// TIA Portal V20 export
FUNCTION_BLOCK "Sensors"   // FB505, FBD
{ S7_Optimized_Access := 'TRUE' }
// stored: AutoNumber false, MemoryReserve 100, SetENOAutomatically false
   VAR
      Var { ExternalAccessible := 'False'; ExternalVisible := 'False'; ExternalWritable := 'False'} : "TypeVar";
      Enc { ExternalAccessible := 'False'; ExternalVisible := 'False'; ExternalWritable := 'False'} : Array[1..3] of "SysCounterFast";
      S { ExternalAccessible := 'False'; ExternalVisible := 'False'; ExternalWritable := 'False'} : Array[1..5] of "SysSensor";
      SIO { ExternalAccessible := 'False'; ExternalVisible := 'False'; ExternalWritable := 'False'} : Array[1..3] of "SysWenglorP3PC301";
      senRightEncAct { ExternalAccessible := 'False'; ExternalVisible := 'False'; ExternalWritable := 'False'} : Real;
      senRightValSmoth { ExternalAccessible := 'False'; ExternalVisible := 'False'; ExternalWritable := 'False'} : Real;
      senRightCntr { ExternalAccessible := 'False'; ExternalVisible := 'False'; ExternalWritable := 'False'} : DInt;
      senRightSum { ExternalAccessible := 'False'; ExternalVisible := 'False'; ExternalWritable := 'False'} : Real;
      senLeftEncAct { ExternalAccessible := 'False'; ExternalVisible := 'False'; ExternalWritable := 'False'} : Real;
      senLeftValSmoth { ExternalAccessible := 'False'; ExternalVisible := 'False'; ExternalWritable := 'False'} : Real;
      senLeftCntr { ExternalAccessible := 'False'; ExternalVisible := 'False'; ExternalWritable := 'False'} : DInt;
      senLeftSum { ExternalAccessible := 'False'; ExternalVisible := 'False'; ExternalWritable := 'False'} : Real;
      senTopEncAct { ExternalAccessible := 'False'; ExternalVisible := 'False'; ExternalWritable := 'False'} : Real;
      senTopValSmoth { ExternalAccessible := 'False'; ExternalVisible := 'False'; ExternalWritable := 'False'} : Real;
      senTopCntr { ExternalAccessible := 'False'; ExternalVisible := 'False'; ExternalWritable := 'False'} : DInt;
      senTopSum { ExternalAccessible := 'False'; ExternalVisible := 'False'; ExternalWritable := 'False'} : Real;
      deltaSaved { ExternalAccessible := 'False'; ExternalVisible := 'False'; ExternalWritable := 'False'} : Real;
      senLeftValValid { ExternalAccessible := 'False'; ExternalVisible := 'False'; ExternalWritable := 'False'} : Bool;
      senRightValValid { ExternalAccessible := 'False'; ExternalVisible := 'False'; ExternalWritable := 'False'} : Bool;
      senTopValValid { ExternalAccessible := 'False'; ExternalVisible := 'False'; ExternalWritable := 'False'} : Bool;
      widthMeasureOk { ExternalAccessible := 'False'; ExternalVisible := 'False'; ExternalWritable := 'False'} : Bool;
   END_VAR
   VAR_TEMP
      tempMin : Real;
      tempMax : Real;
      tempWidth : Real;
   END_VAR
   VAR_TEMP   // added for the SCL form of the ladder/FBD networks
      _w1 : Bool;
   END_VAR
BEGIN

REGION Network 1: encoder infeed scanner
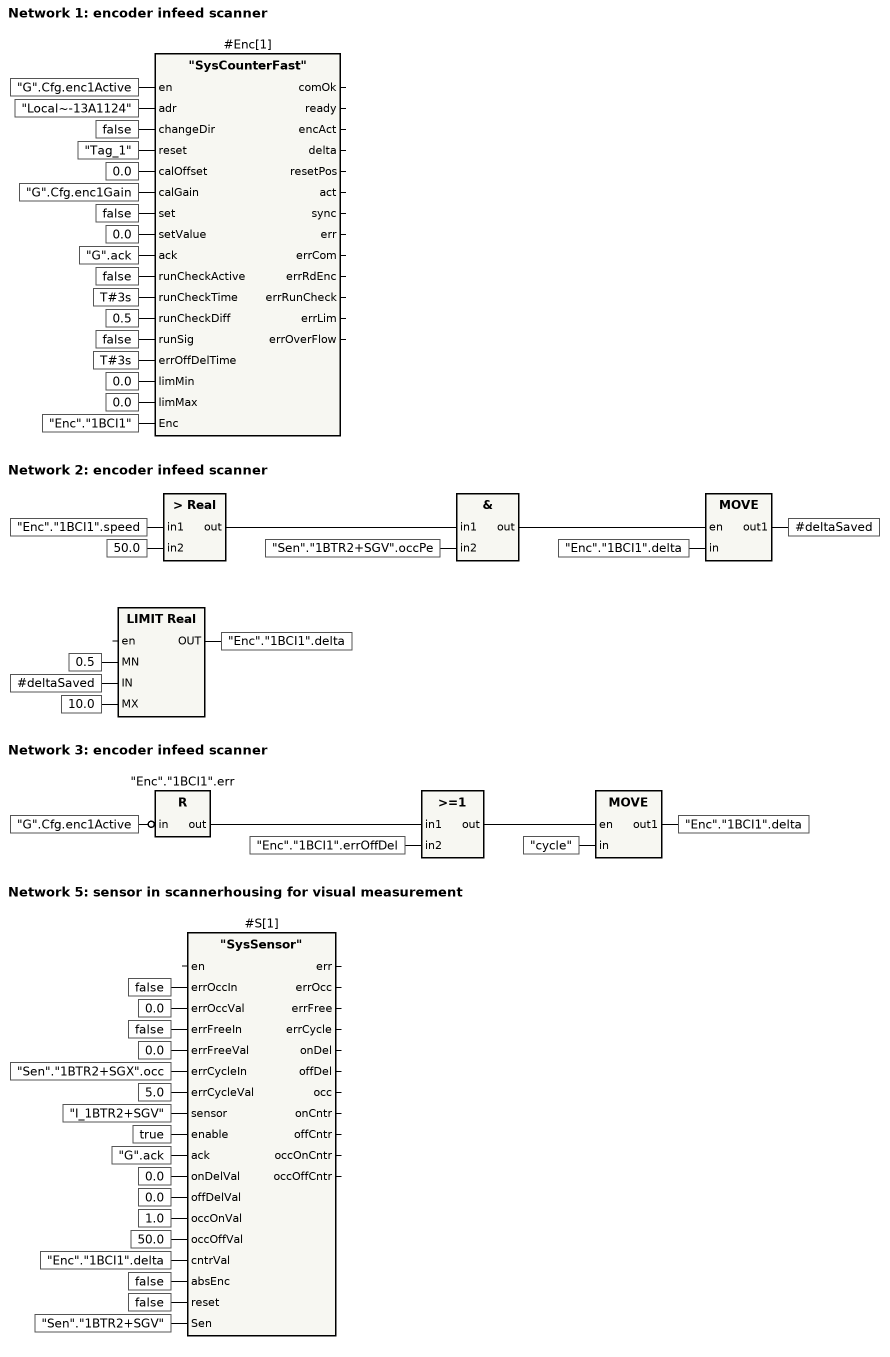
   IF "G".Cfg.enc1Active THEN
       #Enc[1](adr := "Local~-13A1124",   // "SysCounterFast"
               changeDir := false,
               reset := "Tag_1",
               calOffset := 0.0,
               calGain := "G".Cfg.enc1Gain,
               set := false,
               setValue := 0.0,
               ack := "G".ack,
               runCheckActive := false,
               runCheckTime := T#3s,
               runCheckDiff := 0.5,
               runSig := false,
               errOffDelTime := T#3s,
               limMin := 0.0,
               limMax := 0.0,
               Enc := "Enc"."1BCI1");
   END_IF;
END_REGION

REGION Network 2: encoder infeed scanner
   IF ("Enc"."1BCI1".speed > 50.0) AND "Sen"."1BTR2+SGV".occPe THEN
       #deltaSaved := "Enc"."1BCI1".delta;
   END_IF;
   "Enc"."1BCI1".delta := LIMIT(MN := 0.5, IN := #deltaSaved, MX := 10.0);
END_REGION

REGION Network 3: encoder infeed scanner
   IF NOT "G".Cfg.enc1Active THEN "Enc"."1BCI1".err := FALSE; END_IF;
   IF NOT "G".Cfg.enc1Active OR "Enc"."1BCI1".errOffDel THEN "Enc"."1BCI1".delta := "cycle"; END_IF;
END_REGION

REGION Network 4: - sensor monitoring -
END_REGION

REGION Network 5: sensor in scannerhousing for visual measurement
   #S[1](errOccIn := false,   // "SysSensor"
         errOccVal := 0.0,
         errFreeIn := false,
         errFreeVal := 0.0,
         errCycleIn := "Sen"."1BTR2+SGX".occ,
         errCycleVal := 5.0,
         sensor := "I_1BTR2+SGV",
         enable := true,
         ack := "G".ack,
         onDelVal := 0.0,
         offDelVal := 0.0,
         occOnVal := 1.0,
         occOffVal := 50.0,
         cntrVal := "Enc"."1BCI1".delta,
         absEnc := false,
         reset := false,
         Sen := "Sen"."1BTR2+SGV");
END_REGION

REGION Network 6: sensor in scannerhousing for xray measurement
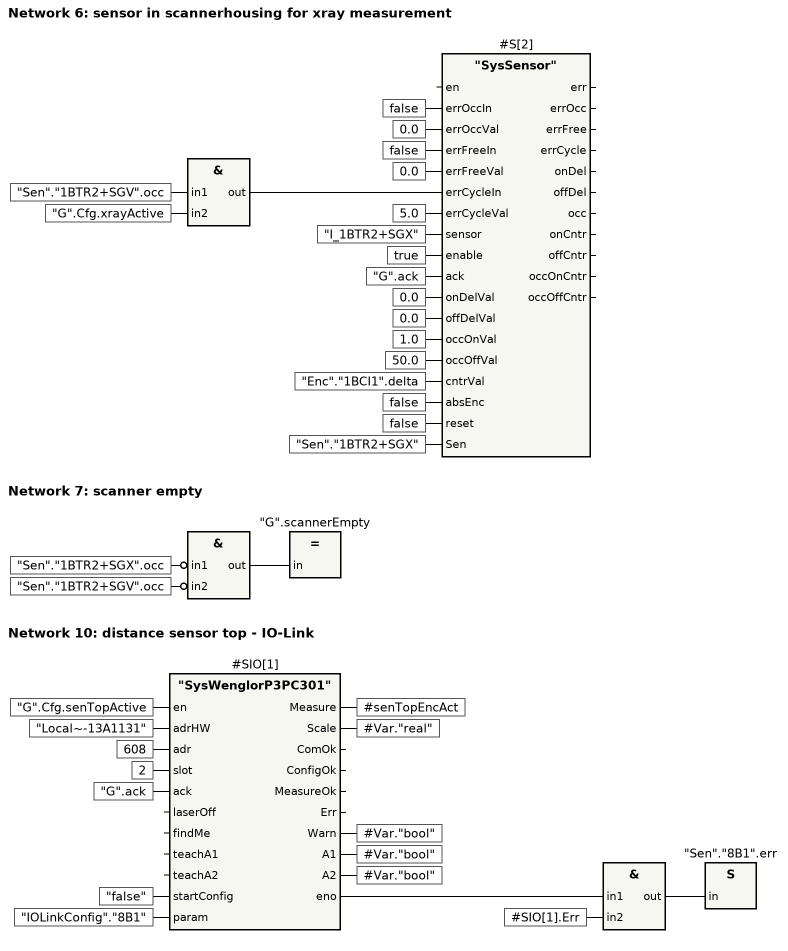
   #S[2](errOccIn := false,   // "SysSensor"
         errOccVal := 0.0,
         errFreeIn := false,
         errFreeVal := 0.0,
         errCycleIn := "Sen"."1BTR2+SGV".occ AND "G".Cfg.xrayActive,
         errCycleVal := 5.0,
         sensor := "I_1BTR2+SGX",
         enable := true,
         ack := "G".ack,
         onDelVal := 0.0,
         offDelVal := 0.0,
         occOnVal := 1.0,
         occOffVal := 50.0,
         cntrVal := "Enc"."1BCI1".delta,
         absEnc := false,
         reset := false,
         Sen := "Sen"."1BTR2+SGX");
END_REGION

REGION Network 7: scanner empty
   "G".scannerEmpty := NOT "Sen"."1BTR2+SGX".occ AND NOT "Sen"."1BTR2+SGV".occ;
END_REGION

REGION Network 8: distance sensor top
END_REGION

REGION Network 9 (SCL): distance sensor top - calibration value from pc
   "ComSd".Data.Measure.SetCalibratePosTopOk := FALSE;

   IF "ComRd".Data.Measure.SetCalibratePosTop THEN

       "Ref".senTopCalOffset := #senTopEncAct + "G".Batch.thickness;
       "ComSd".Data.Measure.SetCalibratePosTopOk := TRUE;
   END_IF;
END_REGION

REGION Network 10: distance sensor top - IO-Link
   #SIO[1](EN := "G".Cfg.senTopActive,   // "SysWenglorP3PC301"
           adrHW := "Local~-13A1131",
           adr := 608,
           slot := 2,
           ack := "G".ack,
           startConfig := "false",
           param := "IOLinkConfig"."8B1",
           Measure => #senTopEncAct,
           Scale => #Var."real",
           Warn => #Var."bool",
           A1 => #Var."bool",
           A2 => #Var."bool",
           ENO => #_w1);
   IF #_w1 AND #SIO[1].Err THEN "Sen"."8B1".err := TRUE; END_IF;
END_REGION

REGION Network 11 (SCL): distance sensor top - values
   IF "G".Cfg.senTopActive THEN
       IF #SIO[1].MeasureOk THEN
           "Sen"."8B1".val := "Ref".senTopCalOffset - #senTopEncAct;
       ELSE
           "Sen"."8B1".val := -50.0;
       END_IF;
       "ComSd".Data.Measure.ActValueTop := REAL_TO_DINT(#senTopEncAct * 10.0);

       IF "G".Cfg.modeBoardPassing = 3 THEN
           #tempMin := "G".Batch.widthMin / 4.0;
           #tempMax := "G".Batch.widthMax + 50.0;
       ELSE
           #tempMin := "G".Batch.widthMin / 2.0;
           #tempMax := "G".Batch.widthMax + 50.0;
       END_IF;
   ELSE
       #senTopEncAct :=  "Sen"."8B1".val := 0.0;
       "ComSd".Data.Measure.ActValueTop := 0;
   END_IF;
END_REGION

REGION Network 12: distance sensor top - occupied
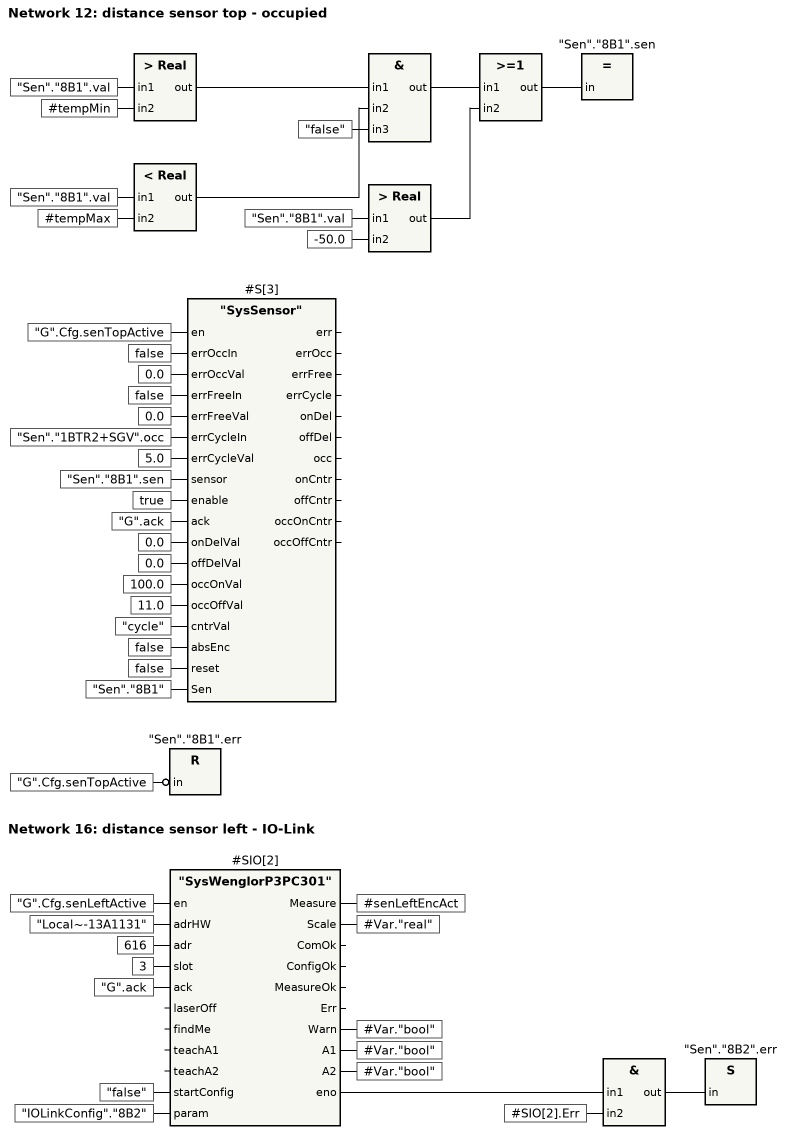
   "Sen"."8B1".sen := (("Sen"."8B1".val > #tempMin) AND ("Sen"."8B1".val < #tempMax) AND "false") OR ("Sen"."8B1".val > (-50.0));
   IF "G".Cfg.senTopActive THEN
       #S[3](errOccIn := false,   // "SysSensor"
             errOccVal := 0.0,
             errFreeIn := false,
             errFreeVal := 0.0,
             errCycleIn := "Sen"."1BTR2+SGV".occ,
             errCycleVal := 5.0,
             sensor := "Sen"."8B1".sen,
             enable := true,
             ack := "G".ack,
             onDelVal := 0.0,
             offDelVal := 0.0,
             occOnVal := 100.0,
             occOffVal := 11.0,
             cntrVal := "cycle",
             absEnc := false,
             reset := false,
             Sen := "Sen"."8B1");
   END_IF;
   IF NOT "G".Cfg.senTopActive THEN "Sen"."8B1".err := FALSE; END_IF;
END_REGION

REGION Network 13 (SCL): distance sensor top - smoothed value
   IF "Sen"."8B1".occPe THEN
       #senTopCntr := 10;
       #senTopSum := 0.0;
       #senTopValValid := false;
   ELSIF NOT "Sen"."8B1".occ OR #senTopCntr > 10 THEN
       #senTopCntr := 0;
   END_IF;

   IF "Sen"."8B1".occNe THEN
       #senTopValValid := false;
   END_IF;

   IF #senTopCntr > 0 AND "Sen"."8B1".sen THEN
       #senTopSum += "Sen"."8B1".val;
       #senTopCntr -= 1;
       IF #senTopCntr = 0 THEN
           #senTopValSmoth := #senTopSum / 10.0;
           #senTopValValid := true;
       END_IF;
   END_IF;

   IF "ComRd".Data.status.Auto AND  "G".Cfg.senTopActive THEN
       "Sen"."8B1".val := #senTopValSmoth;
   END_IF;
END_REGION

REGION Network 14: distance sensor left
END_REGION

REGION Network 15 (SCL): distance sensor left - calibration value from pc
   "ComSd".Data.Measure.SetCalibratePosLeftOk := FALSE;

   IF "ComRd".Data.Measure.SetCalibratePosLeft THEN

       #tempWidth := "G".Batch.width;
       IF "G".Cfg.modeBoardPassing = 3 THEN
           #tempWidth := "G".Batch.width / 2.0;
       END_IF;
       "Ref".senLeftCalOffset := #senLeftEncAct + #tempWidth;

       "ComSd".Data.Measure.SetCalibratePosLeftOk := TRUE;
   END_IF;
END_REGION

REGION Network 16: distance sensor left - IO-Link
   #SIO[2](EN := "G".Cfg.senLeftActive,   // "SysWenglorP3PC301"
           adrHW := "Local~-13A1131",
           adr := 616,
           slot := 3,
           ack := "G".ack,
           startConfig := "false",
           param := "IOLinkConfig"."8B2",
           Measure => #senLeftEncAct,
           Scale => #Var."real",
           Warn => #Var."bool",
           A1 => #Var."bool",
           A2 => #Var."bool",
           ENO => #_w1);
   IF #_w1 AND #SIO[2].Err THEN "Sen"."8B2".err := TRUE; END_IF;
END_REGION

REGION Network 17 (SCL): distance sensor left - values
   IF "G".Cfg.senLeftActive THEN

       IF #SIO[2].MeasureOk THEN
           "Sen"."8B2".val := "Ref".senLeftCalOffset - #senLeftEncAct;
       ELSE
           "Sen"."8B2".val := -50.0;
       END_IF;
       "ComSd".Data.Measure.ActValueLeft := REAL_TO_DINT("Sen"."8B2".val * 10.0);

       IF "G".Cfg.modeBoardPassing = 3 THEN
           #tempMin := "G".Batch.widthMin / 4.0;
           #tempMax := "G".Batch.widthMax + 50.0;
       ELSE
           #tempMin := "G".Batch.widthMin / 2.0;
           #tempMax := "G".Batch.widthMax + 50.0;
       END_IF;
   ELSE
       #senLeftEncAct :=  "Sen"."8B2".val := 0.0;
       "ComSd".Data.Measure.ActValueLeft := 0;
   END_IF;
END_REGION

REGION Network 18: distance sensor left - occupied
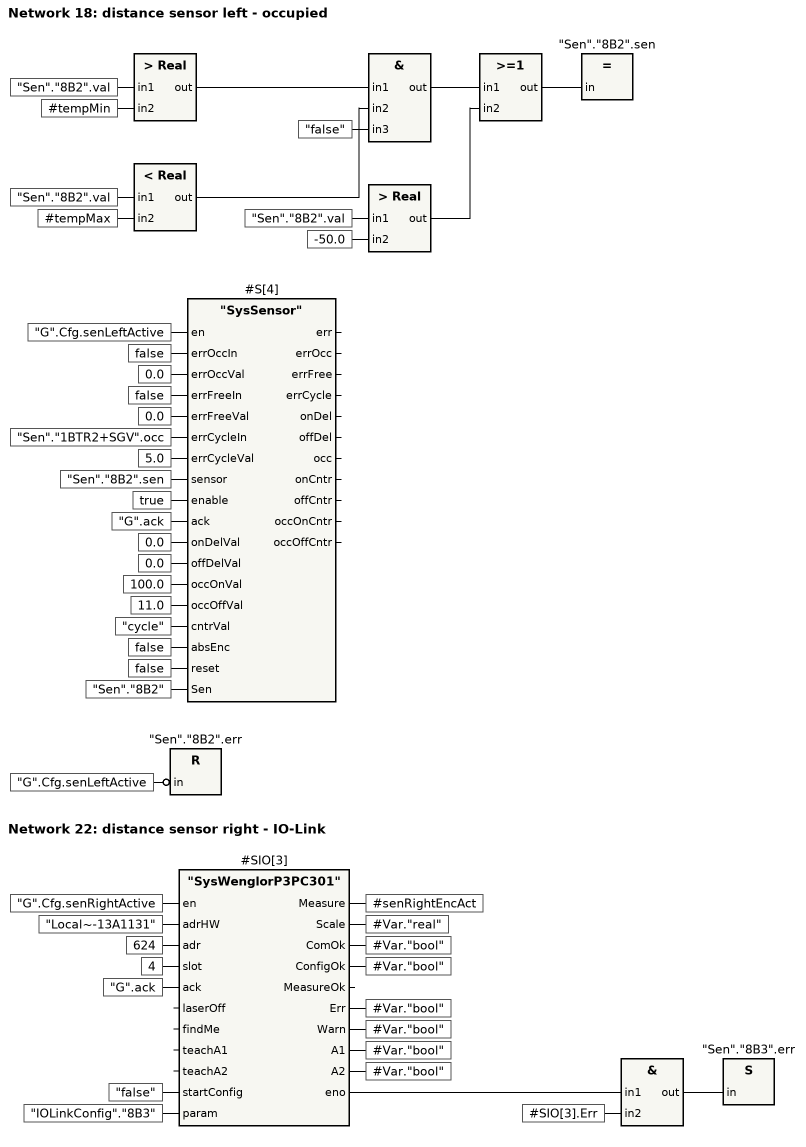
   "Sen"."8B2".sen := (("Sen"."8B2".val > #tempMin) AND ("Sen"."8B2".val < #tempMax) AND "false") OR ("Sen"."8B2".val > (-50.0));
   IF "G".Cfg.senLeftActive THEN
       #S[4](errOccIn := false,   // "SysSensor"
             errOccVal := 0.0,
             errFreeIn := false,
             errFreeVal := 0.0,
             errCycleIn := "Sen"."1BTR2+SGV".occ,
             errCycleVal := 5.0,
             sensor := "Sen"."8B2".sen,
             enable := true,
             ack := "G".ack,
             onDelVal := 0.0,
             offDelVal := 0.0,
             occOnVal := 100.0,
             occOffVal := 11.0,
             cntrVal := "cycle",
             absEnc := false,
             reset := false,
             Sen := "Sen"."8B2");
   END_IF;
   IF NOT "G".Cfg.senLeftActive THEN "Sen"."8B2".err := FALSE; END_IF;
END_REGION

REGION Network 19 (SCL): distance sensor left - smoothed value
   IF "Sen"."8B2".occPe THEN
       #senLeftCntr := 10;
       #senLeftSum := 0.0;
       #senLeftValValid := false;
   ELSIF NOT "Sen"."8B2".occ OR #senLeftCntr > 10 THEN
       #senLeftCntr := 0;
   END_IF;

   IF "Sen"."8B2".occNe THEN
       #senLeftValValid := false;
   END_IF;

   IF #senLeftCntr > 0 AND "Sen"."8B2".sen THEN
       #senLeftSum += "Sen"."8B2".val;
       #senLeftCntr -= 1;
       IF #senLeftCntr = 0 THEN
           #senLeftValSmoth := #senLeftSum / 10.0;
           #senLeftValValid := true;
       END_IF;
   END_IF;

   IF "ComRd".Data.status.Auto AND  "G".Cfg.senLeftActive THEN
       "Sen"."8B2".val := #senLeftValSmoth;
   END_IF;
END_REGION

REGION Network 20: distance sensor right
END_REGION

REGION Network 21 (SCL): distance sensor right - calibration value from pc
   "ComSd".Data.Measure.SetCalibratePosRightOk := FALSE;

   IF "ComRd".Data.Measure.SetCalibratePosRight THEN

       #tempWidth := "G".Batch.width;
       IF "G".Cfg.modeBoardPassing = 3 THEN
           #tempWidth := "G".Batch.width / 2.0;
       END_IF;
       "Ref".senRightCalOffset := #senRightEncAct + #tempWidth;

       "ComSd".Data.Measure.SetCalibratePosRightOk := TRUE;
   END_IF;
END_REGION

REGION Network 22: distance sensor right - IO-Link
   #SIO[3](EN := "G".Cfg.senRightActive,   // "SysWenglorP3PC301"
           adrHW := "Local~-13A1131",
           adr := 624,
           slot := 4,
           ack := "G".ack,
           startConfig := "false",
           param := "IOLinkConfig"."8B3",
           Measure => #senRightEncAct,
           Scale => #Var."real",
           ComOk => #Var."bool",
           ConfigOk => #Var."bool",
           Err => #Var."bool",
           Warn => #Var."bool",
           A1 => #Var."bool",
           A2 => #Var."bool",
           ENO => #_w1);
   IF #_w1 AND #SIO[3].Err THEN "Sen"."8B3".err := TRUE; END_IF;
END_REGION

REGION Network 23 (SCL): distance sensor right - values
   IF "G".Cfg.senRightActive THEN
       IF #SIO[3].MeasureOk THEN
           "Sen"."8B3".val := "Ref".senRightCalOffset - #senRightEncAct;
       ELSE
           "Sen"."8B3".val := -50.0;
       END_IF;
       "ComSd".Data.Measure.ActValueRight := REAL_TO_DINT("Sen"."8B3".val * 10.0);

       IF "G".Cfg.modeBoardPassing = 3 THEN
           #tempMin := "G".Batch.widthMin / 4.0;
           #tempMax := "G".Batch.widthMax + 50.0;
       ELSE
           #tempMin := "G".Batch.widthMin / 2.0;
           #tempMax := "G".Batch.widthMax + 50.0;
       END_IF;
   ELSE
       #senRightEncAct :=  "Sen"."8B3".val := 0.0;
       "ComSd".Data.Measure.ActValueRight := 0;
   END_IF;
END_REGION

REGION Network 24: distance sensor right - occupied
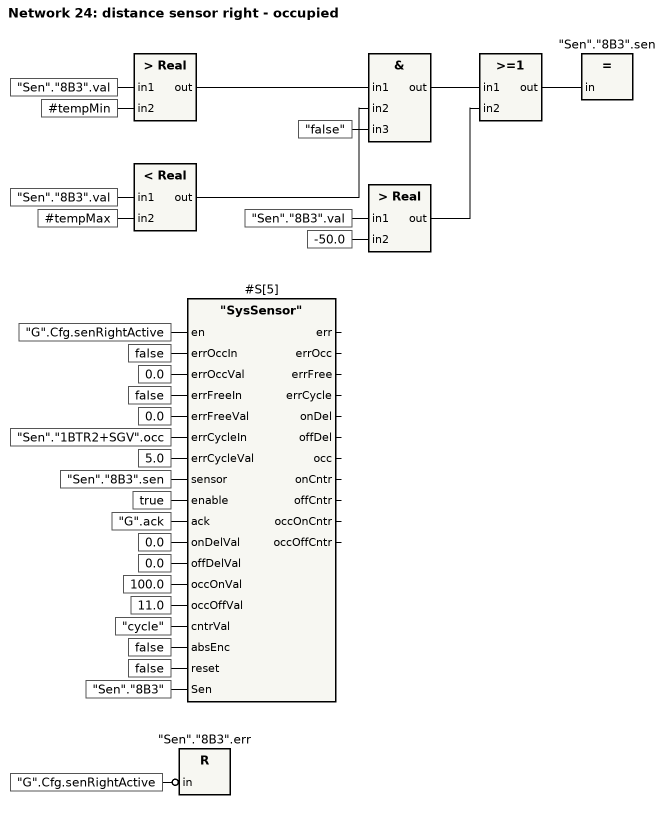
   "Sen"."8B3".sen := (("Sen"."8B3".val > #tempMin) AND ("Sen"."8B3".val < #tempMax) AND "false") OR ("Sen"."8B3".val > (-50.0));
   IF "G".Cfg.senRightActive THEN
       #S[5](errOccIn := false,   // "SysSensor"
             errOccVal := 0.0,
             errFreeIn := false,
             errFreeVal := 0.0,
             errCycleIn := "Sen"."1BTR2+SGV".occ,
             errCycleVal := 5.0,
             sensor := "Sen"."8B3".sen,
             enable := true,
             ack := "G".ack,
             onDelVal := 0.0,
             offDelVal := 0.0,
             occOnVal := 100.0,
             occOffVal := 11.0,
             cntrVal := "cycle",
             absEnc := false,
             reset := false,
             Sen := "Sen"."8B3");
   END_IF;
   IF NOT "G".Cfg.senRightActive THEN "Sen"."8B3".err := FALSE; END_IF;
END_REGION

REGION Network 25 (SCL): distance sensor right - smoothed value
   IF "Sen"."8B3".occPe THEN
       #senRightCntr := 10;
       #senRightSum := 0.0;
       #senRightValValid := false;
   ELSIF NOT "Sen"."8B3".occ OR #senRightCntr > 10 THEN
       #senRightCntr := 0;
   END_IF;

   IF "Sen"."8B3".occNe THEN
       #senRightValValid := false;
   END_IF;

   IF #senRightCntr > 0 AND "Sen"."8B3".sen THEN
       #senRightSum += "Sen"."8B3".val;
       #senRightCntr -= 1;
       IF #senRightCntr = 0 THEN
           #senRightValSmoth := #senRightSum / 10.0;
           #senRightValValid := true;
       END_IF;
   END_IF;

   IF "ComRd".Data.status.Auto AND  "G".Cfg.senRightActive THEN
       "Sen"."8B3".val := #senRightValSmoth;
   END_IF;
END_REGION

REGION Network 26 (SCL): distance sensor - data to pc
   // Thickness
   IF "G".Cfg.modeDimension = 3 OR "G".Cfg.modeDimension = 4 AND  NOT "Sen"."1BTR2+SGV".occ THEN
       "G".Batch.thicknessMeasure := "Sen"."8B1".val;
       // Version 5.13 - Dont look at min or max
       // IF "G".Batch.thicknessMeasure < "G".Batch.thicknessMin OR "G".Batch.thicknessMeasure > "G".Batch.thicknessMax  THEN
       //     "G".Batch.thicknessMeasure := "G".Batch.thickness;
       // END_IF;
       "ComSd".Data.Measure.Thickness := REAL_TO_DINT("G".Batch.thicknessMeasure * 10.0);
   ELSE
       "ComSd".Data.Measure.Thickness := 0;
   END_IF;

   // Width
   IF "G".Cfg.modeDimension = 2 OR "G".Cfg.modeDimension = 4 AND NOT "Sen"."1BTR2+SGV".occ  THEN
       #widthMeasureOk := false;
       IF "G".Cfg.modeBoardPassing = 1 AND  #senRightValValid  THEN
           "G".Batch.widthMeasure := "Sen"."8B3".val;
           #widthMeasureOk := true;
       ELSIF "G".Cfg.modeBoardPassing = 2 AND  #senLeftValValid THEN
           "G".Batch.widthMeasure := "Sen"."8B2".val;
           #widthMeasureOk := true;
       ELSIF "G".Cfg.modeBoardPassing = 3  AND #senLeftValValid  AND #senRightValValid  THEN
           "G".Batch.senLeftVal := "Sen"."8B2".val;
           "G".Batch.senRightVal := "Sen"."8B3".val;
           #widthMeasureOk := true;
           // Version 5.13 - Dont look at min or max
           // IF "G".Batch.senLeftVal < "G".Batch.widthMin / 2.0 - 50.0 OR "G".Batch.senLeftVal > "G".Batch.widthMax / 2.0 + 50.0 OR
           //     "G".Batch.senRightVal < "G".Batch.widthMin / 2.0 - 50.0 OR "G".Batch.senRightVal > "G".Batch.widthMax / 2.0 + 50.0 THEN
           //     "G".Batch.senLeftVal := "G".Batch.senRightVal := "G".Batch.width / 2.0;
           //     #widthMeasureOk := false;
           // END_IF;
           "G".Batch.widthMeasure := "G".Batch.senLeftVal + "G".Batch.senRightVal;
           "G".Batch.offsetBoard := ("G".Batch.senLeftVal - "G".Batch.senRightVal) / 2.0;
       END_IF;
       // Version 5.13 - Dont look at min or max
       // IF "G".Batch.widthMeasure < ("G".Batch.widthMin - 50.0)  OR "G".Batch.widthMeasure > ("G".Batch.widthMax + 50.0) THEN
       //     "G".Batch.widthMeasure := "G".Batch.width;
       //     #widthMeasureOk := false;
       // END_IF;
       "ComSd".Data.Measure.Width := REAL_TO_DINT(("G".Batch.widthMeasure) * 10.0);
   ELSE
       "ComSd".Data.Measure.Width := 0;
   END_IF;
END_REGION
END_FUNCTION_BLOCK
